PROGRAM MAIN
VAR
END_VAR

PRG_INIT();
PRG_MACHINE();

END_PROGRAM

(* stored: Version 1.1.0.1
   POU MAIN: Id {55af0903-9ff0-45b9-8f19-64d30f9df59b}, SpecialFunc None *)
